(* CoDeSys 2.3 export: F_READ_WB_VALVESF_CFG.EXP *)

(* POU FUN/PARAMETERS/F_READ_WB_VALVESF_CFG, ST *)
FUNCTION F_READ_WB_VALVESF_CFG : BOOL
VAR_INPUT
	sHead : STRING;
	rTime : REAL;
END_VAR
VAR_IN_OUT
	stConfig : ST_WB_VALVE_CFG;
	fbIdList : FB_IDLIST;
END_VAR
VAR
END_VAR
stConfig.Cycle    := rTime;
stConfig.TimeMax  := F_IDLIST_GETREAL( CONCAT(sHead, '_TimeMax'   ), fbIdList );
stConfig.PushTime := F_IDLIST_GETREAL( CONCAT(sHead, '_PushTime'  ), fbIdList );
stConfig.PushP    := F_IDLIST_GETREAL( CONCAT(sHead, '_PushPress' ), fbIdList );
stConfig.HP       := F_IDLIST_GETBYTE( CONCAT(sHead, '_HP'        ), fbIdList );
END_FUNCTION
